Fanuc KAREL source: IO0216.compact.KL

PROGRAM IO0216
%STACKSIZE=65535
%PRIORITY=65535
%NOLOCKGROUP
ROUTINE RTEST FROM IO0216
ROUTINE RTEST
VAR
L1 : ARRAY[3] OF INTEGER
L2 : XYZWPR
L3 : JOINTPOS9
L4 : POSITION
U2C_37 : BOOLEAN
U2C_38 : REAL
U2C_39 : REAL
U2C_40 : BOOLEAN
U2C_41 : REAL
BEGIN
U2C_37=TRUE
L1[1]=2
U2C_40=TRUE
U2C_41=1.0
L4=$MNUTOOL[1,1]
END RTEST
BEGIN
RTEST
END IO0216
